(* IEC 61131-3 sources: Lasal/CPU_5344_V01/Class/_AlarmX3ParaDer, 1 file *)

(* ---- _AlarmX3ParaDer.st ---- *)
(*!
<Class
	Name               = "_AlarmX3ParaDer"
	Revision           = "0.0"
	RealtimeTask       = "false"
	CyclicTask         = "false"
	BackgroundTask     = "false"
	DefBackground      = "100 ms"
	Sigmatek           = "false"
	OSInterface        = "false"
	HighPriority       = "false"
	Automatic          = "false"
	UpdateMode         = "Prescan"
	SharedCommandTable = "true"
	Objectsize         = "(300,420)">
	<Channels>
		<Server Name="AlarmActief" Visualized="true" Initialize="false" WriteProtected="false" Retentive="false"/>
		<Server Name="ErrorNr" Visualized="true" Initialize="false" WriteProtected="false" Retentive="false"/>
	</Channels>
	<Network Name="_AlarmX3ParaDer">
		<!-- List of Components in this network -->
		<Components>
			<Object
				Name       = "_base"
				Class      = "_AlarmX3Para"
				Position   = "(218,120)"
				Visualized = "true">
				<Channels>
					<Server Name="ClassSvr"/>
					<Client Name="Acknow"/>
					<Client Name="Config" Value="0"/>
					<Client Name="Group"/>
					<Client Name="Para1"/>
					<Client Name="Para2"/>
					<Client Name="Para3"/>
				</Channels>
			</Object>
		</Components>
		<Comments>
		</Comments>
		<!-- List of Connections in this network -->
		<Connections>
			<Connection Source="this.ClassSvr" Destination="_base.ClassSvr" Vertices="(690,210),(518,210),"/>
			<Connection Source="_base.Config" Destination="this.Config" Vertices="(218,210),(38,210),"/>
			<Connection Source="_base.Acknow" Destination="this.Acknow" Vertices="(218,270),(38,270),"/>
			<Connection Source="_base.Group" Destination="this.Group" Vertices="(218,330),(38,330),"/>
			<Connection Source="_base.Para1" Destination="this.Para1" Vertices="(218,390),(38,390),"/>
			<Connection Source="_base.Para2" Destination="this.Para2" Vertices="(218,450),(38,450),"/>
			<Connection Source="_base.Para3" Destination="this.Para3" Vertices="(218,510),(38,510),"/>
		</Connections>
		<!-- Headerfiles -->
		<Options>
		</Options>
	</Network>
</Class>
*)
#pragma using _AlarmX3Para

_AlarmX3ParaDer : CLASS
: _AlarmX3Para
  //Servers:
	AlarmActief 	: SvrCh_DINT;
	ErrorNr 	: SvrCh_DINT;
  //Clients:
  //Variables:
  //Functions:

	FUNCTION VIRTUAL GLOBAL AlarmActief::Read
		VAR_OUTPUT
			output (EAX) 	: DINT;
		END_VAR;

	FUNCTION VIRTUAL GLOBAL AlarmActief::Write
		VAR_INPUT
			input (EAX) 	: DINT;
		END_VAR
		VAR_OUTPUT
			result (EAX) 	: DINT;
		END_VAR;

	FUNCTION VIRTUAL GLOBAL ErrorNr::Write
		VAR_INPUT
			input (EAX) 	: DINT;
		END_VAR
		VAR_OUTPUT
			result (EAX) 	: DINT;
		END_VAR;
  //Tables:
	FUNCTION @STD
		VAR_OUTPUT
			ret_code	: CONFSTATES;
		END_VAR;
	FUNCTION GLOBAL TAB @CT_;
END_CLASS;

FUNCTION VIRTUAL GLOBAL _AlarmX3ParaDer::AlarmActief::Read
	VAR_OUTPUT
		output (EAX) 	: DINT;
	END_VAR

  AlarmActief := ClassSvr;
  Para1 := Para1.Read();
  ErrorNr := Para1;
  if ErrorNr <> 0 then
    AlarmActief := 1;
  end_if;

	output := AlarmActief;

END_FUNCTION

FUNCTION VIRTUAL GLOBAL _AlarmX3ParaDer::AlarmActief::Write
	VAR_INPUT
		input (EAX) 	: DINT;
	END_VAR
	VAR_OUTPUT
		result (EAX) 	: DINT;
	END_VAR

	AlarmActief := input;
  ClassSvr.Write(input:=AlarmActief); //JdK 6-8-2019: also write to classSvr, because classSvr handles alarm to screen
  if IsClientConnected(#Para1) then
    Para1 := Para1.Read();
    ErrorNr := Para1;
  else
    Para1 := ErrorNr;
  end_if;
	result := AlarmActief;

END_FUNCTION

FUNCTION VIRTUAL GLOBAL _AlarmX3ParaDer::ErrorNr::Write
	VAR_INPUT
		input (EAX) 	: DINT;
	END_VAR
	VAR_OUTPUT
		result (EAX) 	: DINT;
	END_VAR

	ErrorNr := input;
  Para1 := ErrorNr;
	result := ErrorNr;

END_FUNCTION
